FUNCTION_BLOCK LaserSensor
  (* Standard: 61499-2 *)
  (* Version 0.1, 2015-00-08, SYY, SYY-PC *)
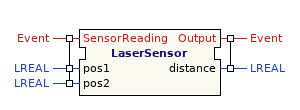
  EVENT_INPUT
    SensorReading WITH pos1, pos2;
  END_EVENT
  EVENT_OUTPUT
    Output WITH distance;
  END_EVENT
  VAR_INPUT
    pos1 : LREAL;
    pos2 : LREAL;
  END_VAR
  VAR_OUTPUT
    distance : LREAL;
  END_VAR
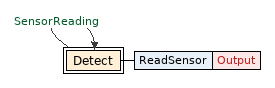
  EC_STATES
    Detect : ReadSensor -> Output;
  END_STATES
  EC_TRANSITIONS
    Detect TO Detect := SensorReading;
  END_TRANSITIONS
  ALGORITHM ReadSensor IN C:
me->distance = me->pos1 - me->pos2;
if(me->distance==0){
me->distance = 100;
}
  END_ALGORITHM
END_FUNCTION_BLOCK
